# EPICS substitutions: IOCs/12id/iocBoot/ioc12idc/quadEM_pid.substitutions
file "$(STD)/stdApp/Db/fast_pid_control.db"
{
pattern
{P,         PID,            INPUT, ICHAN, OUTPUT, OCHAN,    LOPR,     HOPR,  DRVL,  DRVH,  PREC,   KP,    KI,  KD,   DT,        SCAN}
{12idc:, quadEMVertical,    quadEM1,     8,   DAC1,     2,  -32767,    32767,     0,  4095,     3,  .02,  100.,  0., .001, ".1 second"}
{12idc:, quadEMHorizontal,  quadEM1,     9,   DAC1,     3,  -32767,    32767,  2048,  3072,     3,  .02,  100.,  0., .001, ".1 second"}
}
